# EPICS autosave request: galilDmc30017App/Db/galil_dmc30017_analog_in.req
# The files listed here are located at <GALIL support top>/GalilSup/Db
# as they are provided by the Galil Support Module

# All Analog inputs
file "galil_analog_in.req" P=$(P), R=$(ANALOG_IN0)
file "galil_analog_in.req" P=$(P), R=$(ANALOG_IN1)
